FUNCTION_BLOCK TwoCylDiscr
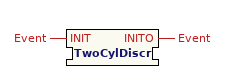
  EVENT_INPUT
    INIT;
  END_EVENT
  EVENT_OUTPUT
    INITO;
  END_EVENT
  FBS
    FB1 : CylControl;
    FB2 : CylControl;
    FB3 : ButtonDs;
    FB4 : LinearDA;
    FB5 : LinearDA;
  END_FBS
  EVENT_CONNECTIONS
    FB3.INITO TO FB4.INIT;
    FB4.INITO TO FB5.INIT;
    FB5.INITO TO FB1.INIT;
    FB1.CNF TO FB4.REQ;
    FB4.CHG TO FB1.REQ;
    FB5.CHG TO FB2.REQ;
    FB1.INITO TO FB2.INIT;
    FB2.CNF TO FB5.REQ;
    FB3.CHG TO FB2.REQ;
    INIT TO FB3.INIT;
    FB2.INITO TO INITO;
    FB3.CHG TO FB1.REQ;
    FB2.INITO TO FB3.REQ;
  END_CONNECTIONS
  DATA_CONNECTIONS
    FB4.HOME TO FB1.Retracted;
    FB4.END TO FB1.Extended;
    FB3.Pressed TO FB1.START;
    FB1.EXTEND TO FB4.FWD;
    FB1.RETRACT TO FB4.BACK;
    FB5.HOME TO FB2.Retracted;
    FB5.END TO FB2.Extended;
    FB2.RETRACT TO FB5.BACK;
    FB2.EXTEND TO FB5.FWD;
    FB3.Pressed TO FB2.START;
  END_CONNECTIONS
END_FUNCTION_BLOCK
